{attribute 'GeneratedUsingTerminal: CU1521-0010-0000'}
{attribute addProperty BoxType "CU1521-0010-0000"}
{attribute addProperty Description "CU1521-0010 EtherCAT media converter (Singlemode)"}
{attribute addProperty Physics "YY"}
{attribute addProperty Id "InfoDataAT %I*InfoData_6F19DB2B2"}
{attribute addProperty CRC "532711307"}
{attribute addProperty Size "2"}
TYPE CU1521_1FC0878B EXTENDS EtcSlaveBoxBase_77A0E4A7 :
STRUCT
	{attribute addProperty Name "InfoData"}
	InfoData : InfoData_6F19DB2B;
END_STRUCT
END_TYPE

(* stored: Version 1.2.0.0, ProductVersion 3.1.4024.9
   DUT CU1521_1FC0878B: Id {e2d94ed7-bb25-4656-922f-f453d09c96dc} *)
